FUNCTION_BLOCK FB_CalculateSiliconThickness
VAR
END_VAR


METHOD PUBLIC Calculate
VAR_INPUT
    fDesiredTransmission : LREAL; // [1]
    fPhotonEnergy : LREAL; // [eV]
END_VAR
VAR_OUTPUT
    fThickness : LREAL; // [mm]
END_VAR
END_METHOD

END_FUNCTION_BLOCK

(* stored: Version 1.1.0.1
   POU FB_CalculateSiliconThickness: Id {ef8c3797-4c77-4129-81d2-4d0dca445cec}, SpecialFunc None
   Method Calculate: Id {23ca27bf-dc1b-46a3-b6bc-af51cedc5a83} *)
